{attribute 'Tc2GvlVarNames'}
VAR_GLOBAL
	
	sGlobClock_SMH					:STRING(12);
END_VAR

(* stored: Version 1.1.0.1, ProductVersion 3.1.4024.15
   GVL GVL_Times: Id {77799a96-9d5a-452a-9d15-f381d1aa399c} *)
